PROGRAM MAIN
VAR
END_VAR

END_PROGRAM

(* stored: Version 1.1.0.1, ProductVersion 3.1.4024.16
   POU MAIN: Id {9f27ee99-5e43-4376-85cf-16eb6998774d}, SpecialFunc None *)
